{attribute 'qualified_only'}
{attribute 'strict'}
TYPE Mode :
(
	Auto,
	Manual
);
END_TYPE

(* stored: Version 1.1.0.1, ProductVersion 3.1.4022.11
   DUT Mode: Id {2b81037d-11a3-461c-a5e5-aa503c0dc3ba} *)
